// Mitsubishi GX Works2 project: DACDT_2026   PLC: Q06UDEH

// task Task_01 (event TRUE, interval 0, priority 31): POU_01
// task Error_Code (event TRUE, interval 0, priority 31): Error_Code
// task HMI_Conver (event TRUE, interval 0, priority 31): HMI_Conver
// task Control (event TRUE, interval 0, priority 31): Control

PROGRAM POU_01
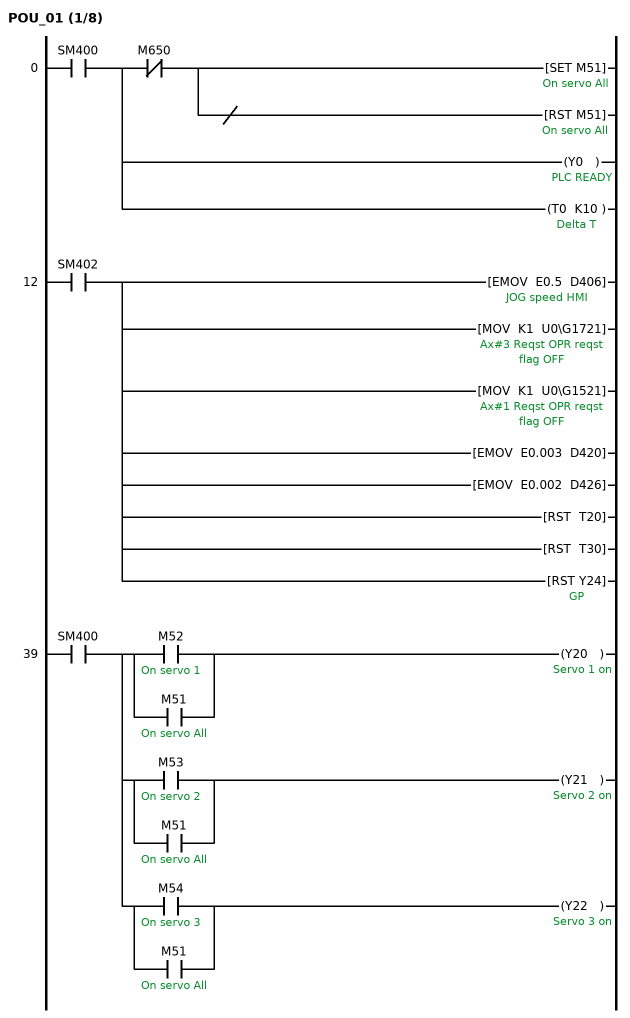
0     LD      SM400
      MPS
      ANI     M650
      SET     M51  ; On servo All
      INV
      RST     M51  ; On servo All
      MPP
      OUT     Y0  ; PLC READY
      OUT     T0 K10  ; Delta T
12    LD      SM402
      EMOV    E0.5 D406  ; JOG speed HMI
      MOV     K1 U0\G1721  ; Ax#3 Reqst OPR reqst flag OFF
      MOV     K1 U0\G1521  ; Ax#1 Reqst OPR reqst flag OFF
      EMOV    E0.003 D420
      EMOV    E0.002 D426
      RST     T20
      RST     T30
      RST     Y24  ; GP
39    LD      SM400
      MPS
      LD      M52  ; On servo 1
      OR      M51  ; On servo All
      ANB
      OUT     Y20  ; Servo 1 on
      MRD
      LD      M53  ; On servo 2
      OR      M51  ; On servo All
      ANB
      OUT     Y21  ; Servo 2 on
      MPP
      LD      M54  ; On servo 3
      OR      M51  ; On servo All
      ANB
      OUT     Y22  ; Servo 3 on
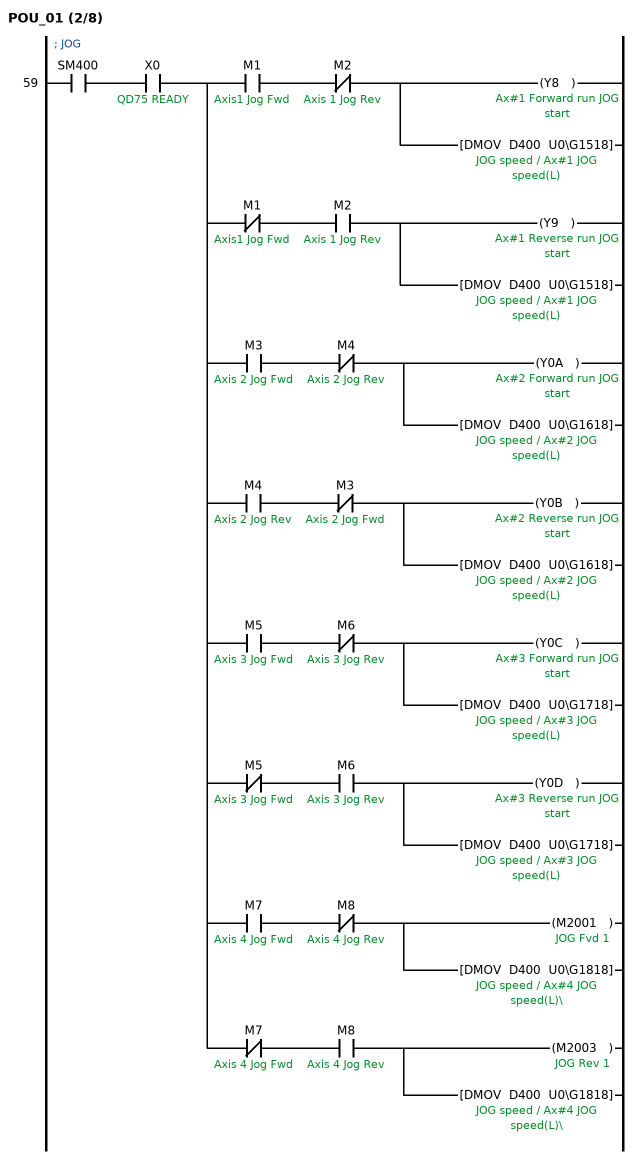
; JOG
59    LD      SM400
      AND     X0  ; QD75 READY
      MPS
      AND     M1  ; Axis1 Jog Fwd
      ANI     M2  ; Axis 1 Jog Rev
      OUT     Y8  ; Ax#1 Forward run JOG start
      DMOV    D400 U0\G1518  ; JOG speed / Ax#1 JOG speed(L)
      MRD
      ANI     M1  ; Axis1 Jog Fwd
      AND     M2  ; Axis 1 Jog Rev
      OUT     Y9  ; Ax#1 Reverse run JOG start
      DMOV    D400 U0\G1518
      MRD
      AND     M3  ; Axis 2 Jog Fwd
      ANI     M4  ; Axis 2 Jog Rev
      OUT     Y0A  ; Ax#2 Forward run JOG start
      DMOV    D400 U0\G1618  ; Ax#2 JOG speed(L)
      MRD
      AND     M4  ; Axis 2 Jog Rev
      ANI     M3  ; Axis 2 Jog Fwd
      OUT     Y0B  ; Ax#2 Reverse run JOG start
      DMOV    D400 U0\G1618
      MRD
      AND     M5  ; Axis 3 Jog Fwd
      ANI     M6  ; Axis 3 Jog Rev
      OUT     Y0C  ; Ax#3 Forward run JOG start
      DMOV    D400 U0\G1718  ; Ax#3 JOG speed(L)
      MRD
      ANI     M5  ; Axis 3 Jog Fwd
      AND     M6  ; Axis 3 Jog Rev
      OUT     Y0D  ; Ax#3 Reverse run JOG start
      DMOV    D400 U0\G1718
      MRD
      AND     M7  ; Axis 4 Jog Fwd
      ANI     M8  ; Axis 4 Jog Rev
      OUT     M2001  ; JOG Fvd 1
      DMOV    D400 U0\G1818  ; Ax#4 JOG speed(L)\
      MPP
      ANI     M7  ; Axis 4 Jog Fwd
      AND     M8  ; Axis 4 Jog Rev
      OUT     M2003  ; JOG Rev 1
      DMOV    D400 U0\G1818
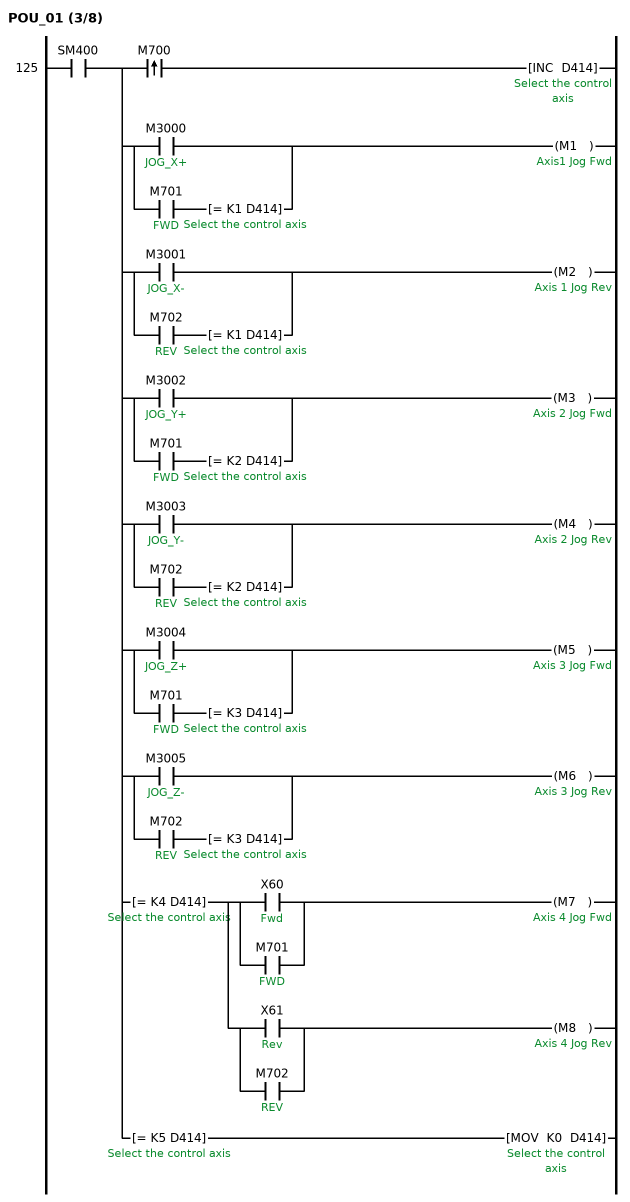
125   LD      SM400
      MPS
      ANDP    M700
      INC     D414  ; Select the control axis
      MRD
      LD      M3000  ; JOG_X+
      LD      M701  ; FWD
      AND=    K1 D414  ; Select the control axis
      ORB
      ANB
      OUT     M1  ; Axis1 Jog Fwd
      MRD
      LD      M3001  ; JOG_X-
      LD      M702  ; REV
      AND=    K1 D414  ; Select the control axis
      ORB
      ANB
      OUT     M2  ; Axis 1 Jog Rev
      MRD
      LD      M3002  ; JOG_Y+
      LD      M701  ; FWD
      AND=    K2 D414  ; Select the control axis
      ORB
      ANB
      OUT     M3  ; Axis 2 Jog Fwd
      MRD
      LD      M3003  ; JOG_Y-
      LD      M702  ; REV
      AND=    K2 D414  ; Select the control axis
      ORB
      ANB
      OUT     M4  ; Axis 2 Jog Rev
      MRD
      LD      M3004  ; JOG_Z+
      LD      M701  ; FWD
      AND=    K3 D414  ; Select the control axis
      ORB
      ANB
      OUT     M5  ; Axis 3 Jog Fwd
      MRD
      LD      M3005  ; JOG_Z-
      LD      M702  ; REV
      AND=    K3 D414  ; Select the control axis
      ORB
      ANB
      OUT     M6  ; Axis 3 Jog Rev
      MRD
      AND=    K4 D414  ; Select the control axis
      MPS
      LD      X60  ; Fwd
      OR      M701  ; FWD
      ANB
      OUT     M7  ; Axis 4 Jog Fwd
      MPP
      LD      X61  ; Rev
      OR      M702  ; REV
      ANB
      OUT     M8  ; Axis 4 Jog Rev
      MPP
      AND=    K5 D414  ; Select the control axis
      MOV     K0 D414
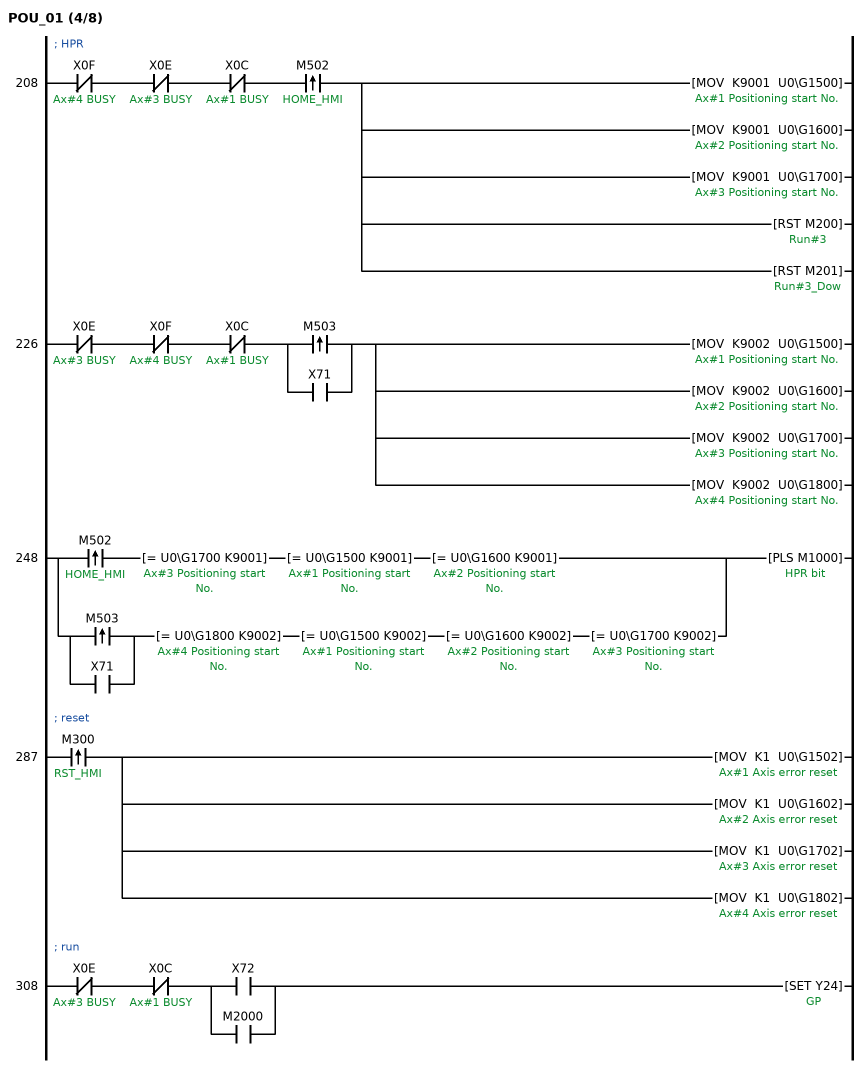
; HPR
208   LDI     X0F  ; Ax#4 BUSY
      ANI     X0E  ; Ax#3 BUSY
      ANI     X0C  ; Ax#1 BUSY
      ANDP    M502  ; HOME_HMI
      MOV     K9001 U0\G1500  ; Ax#1 Positioning start No.
      MOV     K9001 U0\G1600  ; Ax#2 Positioning start No.
      MOV     K9001 U0\G1700  ; Ax#3 Positioning start No.
      RST     M200  ; Run#3
      RST     M201  ; Run#3_Dow
226   LDI     X0E  ; Ax#3 BUSY
      ANI     X0F  ; Ax#4 BUSY
      ANI     X0C  ; Ax#1 BUSY
      LDP     M503
      OR      X71
      ANB
      MOV     K9002 U0\G1500
      MOV     K9002 U0\G1600
      MOV     K9002 U0\G1700
      MOV     K9002 U0\G1800  ; Ax#4 Positioning start No.
248   LDP     M502  ; HOME_HMI
      AND=    U0\G1700 K9001  ; Ax#3 Positioning start No.
      AND=    U0\G1500 K9001  ; Ax#1 Positioning start No.
      AND=    U0\G1600 K9001  ; Ax#2 Positioning start No.
      LDP     M503
      OR      X71
      AND=    U0\G1800 K9002  ; Ax#4 Positioning start No.
      AND=    U0\G1500 K9002  ; Ax#1 Positioning start No.
      AND=    U0\G1600 K9002  ; Ax#2 Positioning start No.
      AND=    U0\G1700 K9002  ; Ax#3 Positioning start No.
      ORB
      PLS     M1000  ; HPR bit
; reset
287   LDP     M300  ; RST_HMI
      MOV     K1 U0\G1502  ; Ax#1 Axis error reset
      MOV     K1 U0\G1602  ; Ax#2 Axis error reset
      MOV     K1 U0\G1702  ; Ax#3 Axis error reset
      MOV     K1 U0\G1802  ; Ax#4 Axis error reset
; run
308   LDI     X0E  ; Ax#3 BUSY
      ANI     X0C  ; Ax#1 BUSY
      LD      X72
      OR      M2000
      ANB
      SET     Y24  ; GP
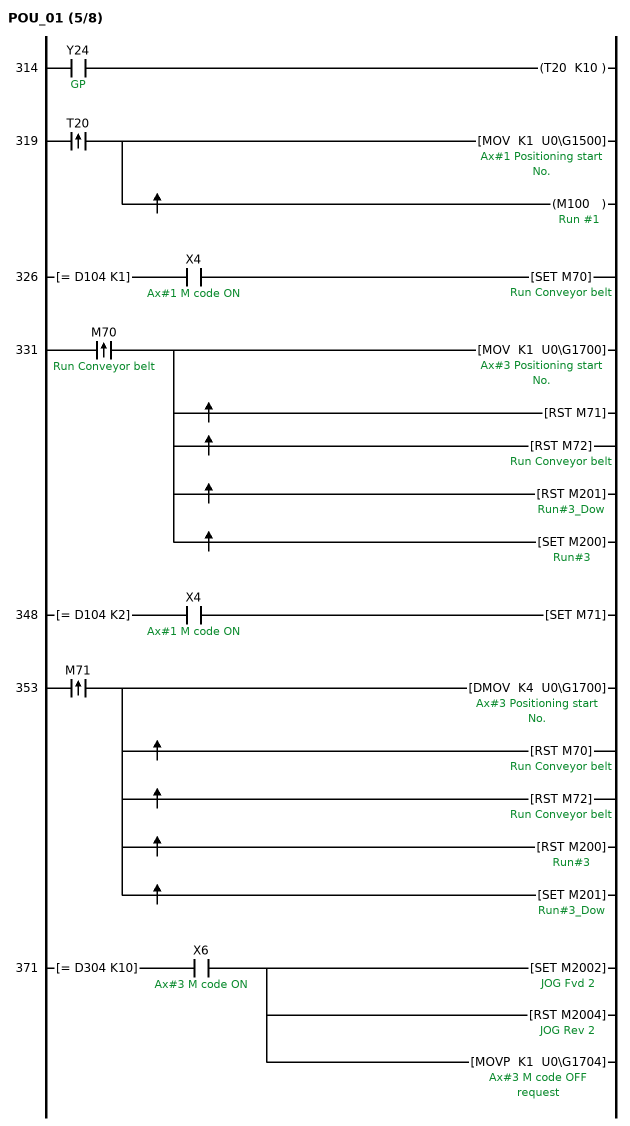
314   LD      Y24  ; GP
      OUT     T20 K10
319   LDP     T20
      MOV     K1 U0\G1500
      MEP
      OUT     M100  ; Run #1
326   LD=     D104 K1
      AND     X4  ; Ax#1 M code ON
      SET     M70  ; Run Conveyor belt
331   LDP     M70  ; Run Conveyor belt
      MOV     K1 U0\G1700
      MPS
      MEP
      RST     M71
      MRD
      MEP
      RST     M72  ; Run Conveyor belt
      MRD
      MEP
      RST     M201  ; Run#3_Dow
      MPP
      MEP
      SET     M200  ; Run#3
348   LD=     D104 K2
      AND     X4  ; Ax#1 M code ON
      SET     M71
353   LDP     M71
      DMOV    K4 U0\G1700
      MPS
      MEP
      RST     M70  ; Run Conveyor belt
      MRD
      MEP
      RST     M72  ; Run Conveyor belt
      MRD
      MEP
      RST     M200  ; Run#3
      MPP
      MEP
      SET     M201  ; Run#3_Dow
371   LD=     D304 K10
      AND     X6  ; Ax#3 M code ON
      SET     M2002  ; JOG Fvd 2
      RST     M2004  ; JOG Rev 2
      MOVP    K1 U0\G1704  ; Ax#3 M code OFF request
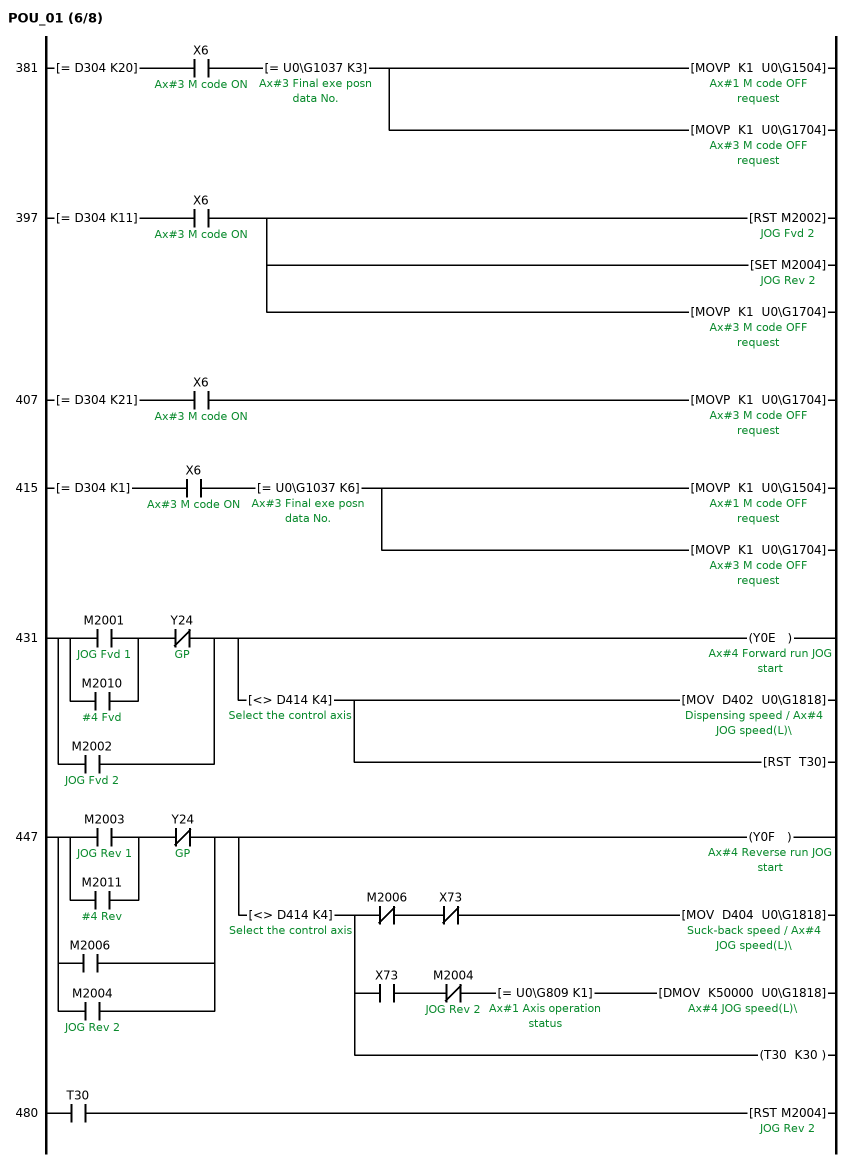
381   LD=     D304 K20
      AND     X6  ; Ax#3 M code ON
      AND=    U0\G1037 K3  ; Ax#3 Final exe posn data No.
      MOVP    K1 U0\G1504  ; Ax#1 M code OFF request
      MOVP    K1 U0\G1704
397   LD=     D304 K11
      AND     X6  ; Ax#3 M code ON
      RST     M2002  ; JOG Fvd 2
      SET     M2004  ; JOG Rev 2
      MOVP    K1 U0\G1704
407   LD=     D304 K21
      AND     X6  ; Ax#3 M code ON
      MOVP    K1 U0\G1704
415   LD=     D304 K1
      AND     X6  ; Ax#3 M code ON
      AND=    U0\G1037 K6  ; Ax#3 Final exe posn data No.
      MOVP    K1 U0\G1504
      MOVP    K1 U0\G1704
431   LD      M2001  ; JOG Fvd 1
      OR      M2010  ; #4 Fvd
      ANI     Y24  ; GP
      OR      M2002  ; JOG Fvd 2
      OUT     Y0E  ; Ax#4 Forward run JOG start
      AND<>   D414 K4  ; Select the control axis
      MOV     D402 U0\G1818  ; Dispensing speed
      RST     T30
447   LD      M2003  ; JOG Rev 1
      OR      M2011  ; #4 Rev
      ANI     Y24  ; GP
      OR      M2006
      OR      M2004  ; JOG Rev 2
      OUT     Y0F  ; Ax#4 Reverse run JOG start
      AND<>   D414 K4  ; Select the control axis
      MPS
      ANI     M2006
      ANI     X73
      MOV     D404 U0\G1818  ; Suck-back speed
      MRD
      AND     X73
      ANI     M2004  ; JOG Rev 2
      AND=    U0\G809 K1  ; Ax#1 Axis operation status
      DMOV    K50000 U0\G1818
      MPP
      OUT     T30 K30
480   LD      T30
      RST     M2004  ; JOG Rev 2
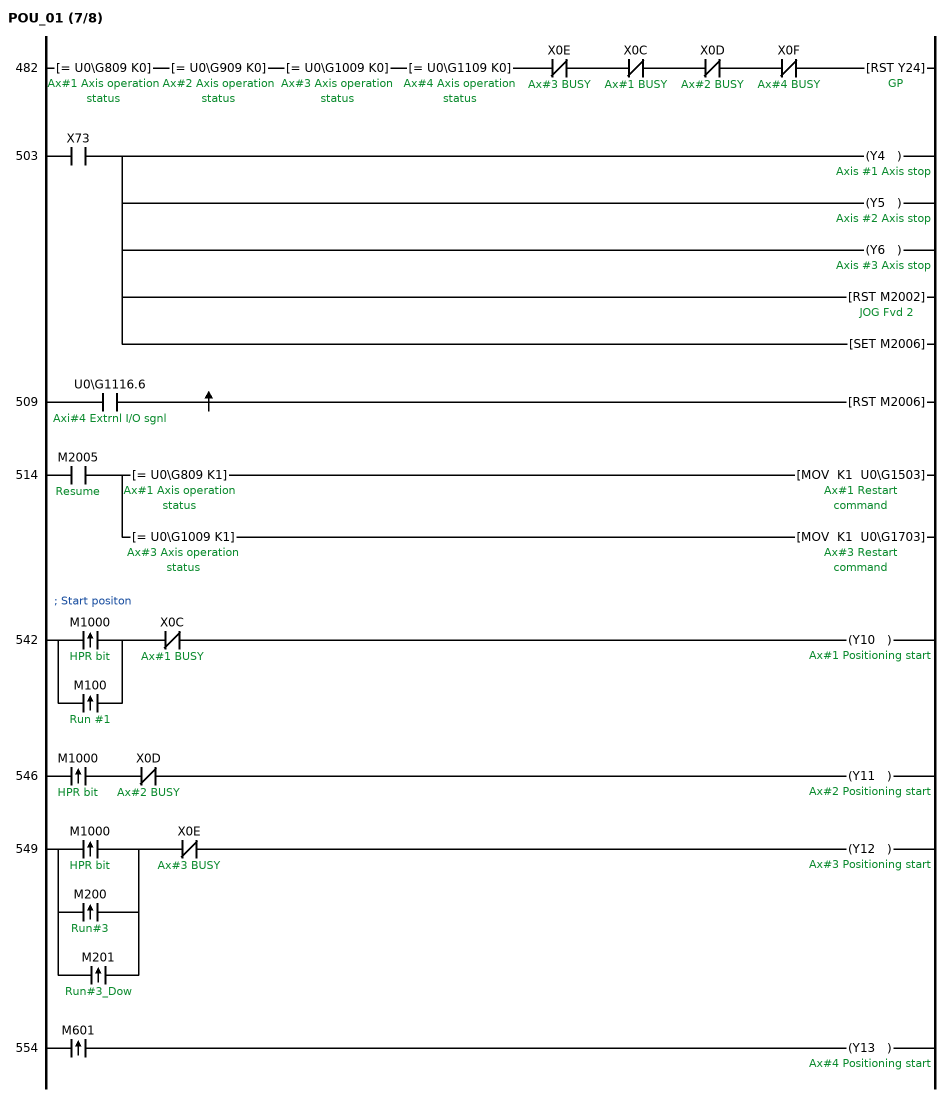
482   LD=     U0\G809 K0  ; Ax#1 Axis operation status
      AND=    U0\G909 K0  ; Ax#2 Axis operation status
      AND=    U0\G1009 K0  ; Ax#3 Axis operation status
      AND=    U0\G1109 K0  ; Ax#4 Axis operation status
      ANI     X0E  ; Ax#3 BUSY
      ANI     X0C  ; Ax#1 BUSY
      ANI     X0D  ; Ax#2 BUSY
      ANI     X0F  ; Ax#4 BUSY
      RST     Y24  ; GP
503   LD      X73
      OUT     Y4  ; Axis #1 Axis stop
      OUT     Y5  ; Axis #2 Axis stop
      OUT     Y6  ; Axis #3 Axis stop
      RST     M2002  ; JOG Fvd 2
      SET     M2006
509   LD      U0\G1116.6  ; Axi#4 Extrnl I/O sgnl
      MEP
      RST     M2006
514   LD      M2005  ; Resume
      MPS
      AND=    U0\G809 K1  ; Ax#1 Axis operation status
      MOV     K1 U0\G1503  ; Ax#1 Restart command
      MPP
      AND=    U0\G1009 K1  ; Ax#3 Axis operation status
      MOV     K1 U0\G1703  ; Ax#3 Restart command
; Start positon
542   LDP     M1000  ; HPR bit
      ORP     M100  ; Run #1
      ANI     X0C  ; Ax#1 BUSY
      OUT     Y10  ; Ax#1 Positioning start
546   LDP     M1000  ; HPR bit
      ANI     X0D  ; Ax#2 BUSY
      OUT     Y11  ; Ax#2 Positioning start
549   LDP     M1000  ; HPR bit
      ORP     M200  ; Run#3
      ORP     M201  ; Run#3_Dow
      ANI     X0E  ; Ax#3 BUSY
      OUT     Y12  ; Ax#3 Positioning start
554   LDP     M601
      OUT     Y13  ; Ax#4 Positioning start
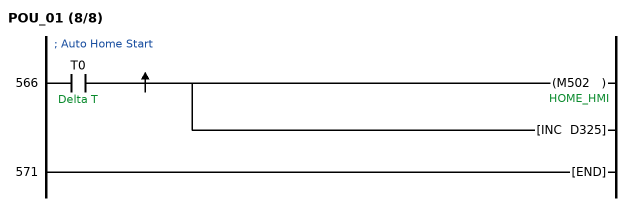
; Auto Home Start
566   LD      T0  ; Delta T
      MEP
      OUT     M502  ; HOME_HMI
      INC     D325
571   END
END_PROGRAM

PROGRAM Error_Code
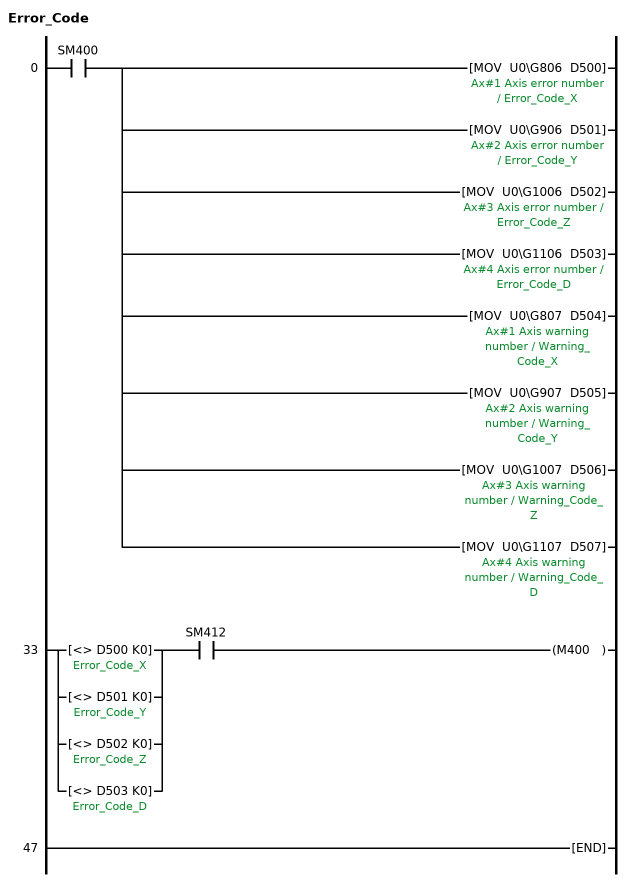
0     LD      SM400
      MOV     U0\G806 D500  ; Ax#1 Axis error number / Error_Code_X
      MOV     U0\G906 D501  ; Ax#2 Axis error number / Error_Code_Y
      MOV     U0\G1006 D502  ; Ax#3 Axis error number / Error_Code_Z
      MOV     U0\G1106 D503  ; Ax#4 Axis error number / Error_Code_D
      MOV     U0\G807 D504  ; Ax#1 Axis warning number / Warning_Code_X
      MOV     U0\G907 D505  ; Ax#2 Axis warning number / Warning_Code_Y
      MOV     U0\G1007 D506  ; Ax#3 Axis warning number / Warning_Code_Z
      MOV     U0\G1107 D507  ; Ax#4 Axis warning number / Warning_Code_D
33    LD<>    D500 K0  ; Error_Code_X
      OR<>    D501 K0  ; Error_Code_Y
      OR<>    D502 K0  ; Error_Code_Z
      OR<>    D503 K0  ; Error_Code_D
      AND     SM412
      OUT     M400
47    END
END_PROGRAM

PROGRAM HMI_Conver
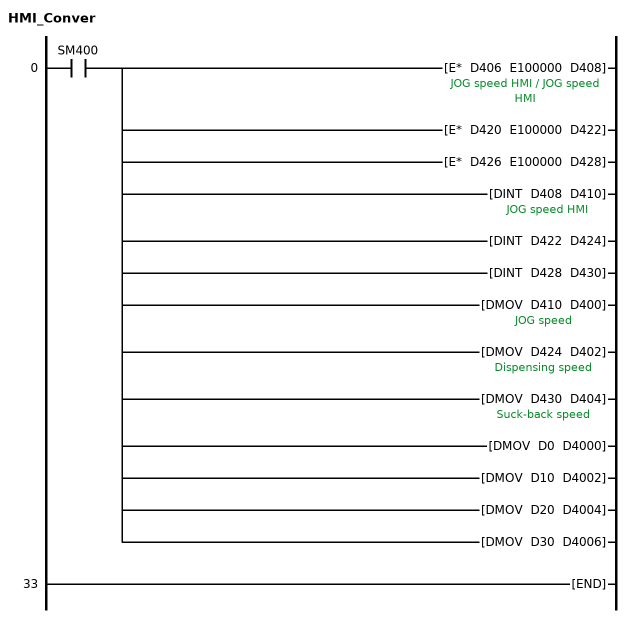
0     LD      SM400
      E*      D406 E100000 D408  ; JOG speed HMI / JOG speed HMI
      E*      D420 E100000 D422
      E*      D426 E100000 D428
      DINT    D408 D410
      DINT    D422 D424
      DINT    D428 D430
      DMOV    D410 D400  ; JOG speed
      DMOV    D424 D402  ; Dispensing speed
      DMOV    D430 D404  ; Suck-back speed
      DMOV    D0 D4000
      DMOV    D10 D4002
      DMOV    D20 D4004
      DMOV    D30 D4006
33    END
END_PROGRAM

PROGRAM Control
IF WORD_TO_INT(D1000) > 0 THEN

    CASE WORD_TO_INT(D1000) OF

        1:(*Đường thẳng*)
        	(*Toạ độ*)
            U0\G2006 := D1100;
            U0\G8006 := D1200;
            (*Speed*)
            U0\G2004 := D1500; 
        2:(*cung tròn CW*)
        
       		(*toạ độ điểm cuối*)
            U0\G2016 := D1100;
            U0\G8016 := D1200;
            (*Toạ độ tâm*)
            U0\G2018 := D1100;
            U0\G8018 := D1200;
            (*Speed*)
            U0\G2004 := D1500;     
            U0\G8004 := D1500;           
        3: (*cung tròn CCW*)
        
			(*toạ độ điểm cuối*)
            U0\G2026 := D1100;
            U0\G8026 := D1200;
            (*Toạ độ tâm*)
            U0\G2028 := D1100;
            U0\G8028 := D1200;
            
            (*Speed*)
            U0\G2004 := D1500;     
            U0\G8004 := D1500;   
        4: (*Hạ trục Z*)

            U0\G14006 := D1100;
             
    END_CASE;

END_IF;
END_PROGRAM

// device comments not shown above
D1000  ; Ma_Lenh
D1100  ; POS_X(micrometer)
D1200  ; POS_Y(micrometer)
D1500  ; Speed(mm\min)
X1  ; Synchronization flag signal
X5  ; Ax#2 M code ON
X7  ; Ax#4 M code ON
X8  ; Ax#1 Error detection
X9  ; Ax#2 Error detection
X0A  ; Ax#3 Error detection
X0B  ; Ax#4 Error detection
X10  ; Ax#1 Start complete
X11  ; Ax#2 Start complete
X12  ; Ax#3 Start complete
X13  ; Ax#4 Start complete
X14  ; Ax#1 Positioning complete
X15  ; Ax#2 Positioning complete
X16  ; Ax#3 Positioning complete
X17  ; Ax#4 Positioning complete
X62  ; On Servo
X63  ; Run
X64  ; S_HPR
X65  ; Stop
X66  ; Select the control axis
X67  ; Run the conveyor
X68  ; Reversing conveyor
X69  ; Turn off conveyor
Y7  ; Axis #4 Axis stop
Y14  ; Ax#1 Exe prhbtn flag sgnl
Y15  ; Ax#2 Exe prhbtn flag sgnl
Y16  ; Ax#3 Exe prhbtn flag sgnl
Y17  ; Ax#4 Exe prhbtn flag sgnl
Y23  ; Open Brk
M0  ; Step On
M30  ; Brk_Axis3
M50  ; Run #3 Down
M55  ; Stop Servo
M56  ; Run Conveyor belt
M57  ; HPR Fast
M58  ; Open Brk
M60  ; Run #3 Down
M61  ; Run #3 up
M62  ; HPR Mcode
M500  ; START_HMI
M501  ; RST_HMI
M600  ; Rset couter
D200  ; #1\2 Speed
D202  ; #3 Speed
D416  ; OPR speed
D418  ; Creep speed
D1300  ; ARC_X(micrometer)
D1400  ; ARC_Y(micrometer)
D1600  ; Dwell_time(ms)
D1700  ; Bit_Run
T10  ; Detal t
